FUNCTION_BLOCK EnhancedAdapterWith (* FB for teseting an adapter WITH connection *)
  (* Standard: 61499-2; Description: Copyright (c) 2023 Johannes Kepler University Linz This program and the accompanying materials are made available under the terms of the Eclipse Public License 2.0 which is available at https://www.eclipse.org/legal/epl-2.0/ SPDX-License-Identifier: EPL-2.0 *)
  (* Version 1.0, 2023-03-08, Bianca Wiesmayr, Johannes Kepler University Linz, initial API and implementation and/or initial documentation *)
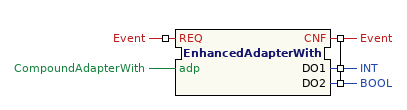
  EVENT_INPUT
    REQ WITH DO1, DO2, DI1, DI2;
  END_EVENT
  EVENT_OUTPUT
    CNF WITH DO1, DO2, DI1, DI2;
  END_EVENT
  VAR_OUTPUT
    DO1 : INT;
    DO2 : BOOL;
  END_VAR
  SOCKETS
    adp : CompoundAdapterWith;
  END_SOCKETS
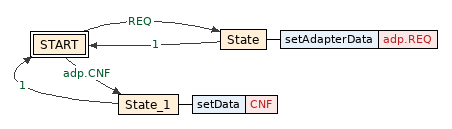
  EC_STATES
    START; (* Initial State *)
    State : setAdapterData -> adp.REQ;
    State_1 : setData -> CNF;
  END_STATES
  EC_TRANSITIONS
    START TO State := REQ;
    State TO START := 1;
    START TO State_1 := adp.CNF;
    State_1 TO START := 1;
  END_TRANSITIONS
  ALGORITHM setAdapterData IN ST:
	adp.DI1 := INT#5;
	adp.DI2 := TRUE;
  END_ALGORITHM
  ALGORITHM setData IN ST:
	DO1 := adp.DO1;
	DO2 := adp.DO2;
  END_ALGORITHM
END_FUNCTION_BLOCK
